INTERFACE I_Entity EXTENDS I_Debug, I_EntityNode

END_INTERFACE

(* stored: Version 1.1.0.1
   Itf I_Entity: Id {77224a92-9fcc-4a74-a8b9-35a817627826} *)
